Staubli VAL3: PickAndPlace1.pjx

--- PickAndPlace1.pjx ---
Parameters version=s7.1 stackSize=5000 millimeterUnit=true
Program file=Pick.pgx
Program file=Place.pgx
Program file=RobotMotion.pgx
Program file=start.pgx
Program file=stop.pgx
Data file=PickAndPlace1.dtx

--- PickAndPlace1.dtx ---
bool bBool1 = true
jointRx jHome
mdesc mNomSpeed
mdesc mSlow = {accel=25, vel=25, decel=25, rmax=25, tmax=25}
num nRep
public pointRx pPointrx1[3]
  [0] = {x=498.015054, y=59.142287, z=-30.989318, rx=5.599382, ry=128.808236, rz=-7.17091, fatherId=world[0]}
  [1] = {x=445.61, y=378.050542, z=199.065349, rx=88.308613, ry=128.361913, rz=-88.673624, fatherId=world[0]}
  [2] = {x=481.810529, y=-248.36011, z=-295.450034, rx=-23.480249, ry=144.718456, rz=48.788162, fatherId=world[0]}
tool tTool1 = {fatherId=flange[0], ioLink=valve1}

--- start.pgx ---
program start()
begin
  call RobotMotion()
end

--- Pick.pgx ---
program Pick(pointRx pPos)
begin
  movel(appro(pPos,{0,0,-50,0,0,0}),tTool1,mNomSpeed)
  delay(3)
  open(tTool1)
  movel(pPos,tTool1,mSlow)
  delay(3)
  close(tTool1)
  movel(appro(pPos,{0,0,-50,0,0,0}),tTool1,mSlow)
  delay(3)
end

--- Place.pgx ---
program Place(pointRx pPos)
begin
  movel(appro(pPos,{0,0,-50,0,0,0}),tTool1,mNomSpeed)
  delay(3)
  movel(appro(pPos,{0,0,-1,0,0,0}),tTool1,mSlow)
  delay(3)
  open(tTool1)
  movel(appro(pPos,{0,0,-50,0,0,0}),tTool1,mSlow)
  delay(3)
  close(tTool1)
end

--- RobotMotion.pgx ---
program RobotMotion()
begin
  movej(jHome,tTool1,mNomSpeed)
  delay(3)
  while (bBool1)
    call Pick(pPointrx1[nRep])
    nRep=nRep+1

    if nRep==3
      nRep=0
      //bBool1.false
    endIf
    call Place(pPointrx1[nRep])
  endWhile
end
